(* CODESYS project TcDynCollections.library
   Company: FisoThemes
   DefaultNamespace: TcDynCollections
   Version: 0.1.0.0
   DocFormat: reStructuredText
   Placeholder: TwinCat Dynamic Collections
   Author: Goodwill Mzumala
   Description: A library for handling collections of data dynamically.
   Title: TwinCat Dynamic Collections

Project tree, tasks and I/O mapping:
  libraries: Tc2_Standard, * (Beckhoff Automation GmbH); Tc2_System, * (Beckhoff Automation GmbH); Tc3_Module, * (Beckhoff Automation GmbH)
  DUTs/
    Interfaces/
      interface I_Collections: _Count, _Error_Status, _Is_Empty, Clear
      interface I_List: Add_Front, Create, FB_exit, FB_init, Get, Get_First, Insert, Remove, RemoveAt, Reverse, Set
      interface I_Queue: Dequeue, Dequeue_Void, Enqueue, Enqueue_At_Front, Peek, Reverse
      interface I_Stack: Peek, Pop, Pop_Void, Push, Top
    Structs/
      data type ST_ERROR
      data type ST_NODE
  GVLs/
  POUs/
    Examples/
      program P_List_Example [ST]
      program P_Queue_Example [ST]
      program P_Stack_Example [ST]
    Function Blocks/
      function block FB_Collections [ST]: _Count, _Error_Status, _Is_Empty, Clear
      function block FB_List [ST]: ClearException, EmptyListException, MemCmpErrExpection, OutOfBoundsException, TypeMismatchException, CopyValueTo, DecrementSize, Free_Node, IncrementSize, Iterate, Malloc_Node, SetValue, _Count, _Is_Empty, Add_Front, Clear, Create, FB_exit, FB_init, Get, Get_First, Insert, Remove, RemoveAt, Reverse, Set
      function block FB_Queue [ST]: _Count, _Is_Empty, CatchError, Clear, Dequeue, Dequeue_Void, Enqueue, Enqueue_At_Front, Peek, Reverse
      function block FB_Stack [ST]: _Count, _Is_Empty, CatchError, Clear, Peek, Pop, Pop_Void, Push, Reverse, Top
    program MAIN [ST]
  Project Information/
    function F_GetCompany [ST]
    function F_GetTitle [ST]
    function F_GetVersion [ST]
  UML/
  Version/
    global variables Global_Version
  VISUs/
*)

// DUTs/Structs/ST_ERROR
(* STRUCT used to contain error status information. *)
{attribute 'enable_dynamic_creation'}
TYPE ST_ERROR :
STRUCT
	bSTATUS : BOOL; 		// Indicates if an error has occurred | TRUE = error, FALSE = no error
	nCODE 	: DINT; 		// Error code specific to the particular error.
	sSOURCE : T_MaxString; 	// Textual information describing the error.
END_STRUCT
END_TYPE

// DUTs/Structs/ST_NODE
{attribute 'enable_dynamic_creation'}
TYPE ST_NODE:
STRUCT
	Data 	: __SYSTEM.AnyType; 							// Stored data.
	sData 	: T_MaxString; 									// Data converted to string.
	pNext 	: POINTER TO ST_NODE := Tc3_Module.GVL.NULL; 	// Pointer to next node. (DEFAULT: NULL pointer)
END_STRUCT
END_TYPE

// Version/Global_Version
{attribute 'TcGenerated'}
{attribute 'no-analysis'}
{attribute 'linkalways'}
// This function has been automatically generated from the project information.
VAR_GLOBAL CONSTANT
	{attribute 'const_non_replaced'}
	stLibVersion_TwinCat_Dynamic_Collections : ST_LibVersion := (iMajor := 0, iMinor := 1, iBuild := 0, iRevision := 0, nFlags := 0, sVersion := '0.1.0.0');
END_VAR

// DUTs/Interfaces/I_Collections
INTERFACE I_Collections

(* Number of elements in collection*)
PROPERTY _Count : DINT
GET
END_GET
END_PROPERTY

(* Gets collection's error status *)
PROPERTY _Error_Status : ST_ERROR
GET
END_GET
END_PROPERTY

(* Checks if collection is empty.*)
PROPERTY _Is_Empty : BOOL
GET
END_GET
END_PROPERTY

(* Empties/Clears/Deletes every element on the collection*)
METHOD Clear
END_METHOD

END_INTERFACE

// DUTs/Interfaces/I_List
INTERFACE I_List EXTENDS I_Collections

// Creates/Adds an node to the front of the list
METHOD Add_Front : I_List
VAR_INPUT
	Value 	: ANY; // Value to store in node
END_VAR
END_METHOD

// Creates/Adds an node to the end of the list
METHOD Create : I_List
VAR_INPUT
	Value 	: ANY; // Value to store in node
END_VAR
END_METHOD

METHOD FB_exit : BOOL
VAR_INPUT
	bInCopyCode : BOOL; // if TRUE, the exit method is called for exiting an instance that is copied afterwards (online change).
END_VAR
END_METHOD

METHOD FB_init : BOOL
VAR_INPUT
	bInitRetains : BOOL; // if TRUE, the retain variables are initialized (warm start / cold start)
	bInCopyCode : BOOL;  // if TRUE, the instance afterwards gets moved into the copy code (online change)
END_VAR
END_METHOD

// Gets value from node at specified location;
METHOD Get : I_List
VAR_INPUT
	Return_Value 	: ANY;  // Variable to store requested node value
	nIndex 			: DINT; // Location of node
END_VAR
END_METHOD

(* Gets value from first node. *) 
METHOD Get_First : I_List
VAR_INPUT
	Return_Value 	: ANY; // Variable to store returned value
END_VAR
END_METHOD

// Adds new node to list at specified location
METHOD Insert : I_List
VAR_INPUT
	Value 	: ANY; // Value to store in node
	nIndex 	: DINT; // Location of node
END_VAR
END_METHOD

(* Removes node at the front of the list and returns nothing. *)
METHOD Remove : I_List
END_METHOD

(* Remove node at specific loacation and return nothing *)
METHOD RemoveAt : I_List
VAR_INPUT
	nIndex : DINT; // Location of node
END_VAR
END_METHOD

// Reverses list
METHOD Reverse : I_List
VAR_INPUT
END_VAR
END_METHOD

// Sets value of node at specified location;
METHOD Set : I_List
VAR_INPUT
	Value 	: ANY; 	// Value to store in node
	nIndex 	: DINT; // Location of node
END_VAR
END_METHOD

END_INTERFACE

// DUTs/Interfaces/I_Queue
INTERFACE I_Queue EXTENDS I_Collections

(* Gets and remove item at the front of the queue *)
METHOD Dequeue : I_Queue
VAR_INPUT
	Item : ANY; (* Variable to store returned item value *)
END_VAR
END_METHOD

(* Removes item at the front of the queue without returning anything *)
METHOD Dequeue_Void : I_Queue
VAR_INPUT
END_VAR
END_METHOD

(* Adds item at the back of the queue *)
METHOD Enqueue : I_Queue
VAR_INPUT
	Item : ANY; (* Variable containg data to store on the queue *)
END_VAR
END_METHOD

(* Adds item at the front of the queue *)
METHOD Enqueue_At_Front : I_Queue
VAR_INPUT
	Item : ANY; (* Variable containg data to store on the queue *)
END_VAR
END_METHOD

(* Get item from the queue without removing it. *)
METHOD Peek : I_Queue
VAR_INPUT
	Item 	: ANY; (* Variable to store returned item value *)
	nIndex 	: DINT; (* Location of item*)
END_VAR
END_METHOD

METHOD Reverse : I_Queue
VAR_INPUT
END_VAR
END_METHOD

END_INTERFACE

// DUTs/Interfaces/I_Stack
INTERFACE I_Stack EXTENDS I_Collections

(* Get item from stack without removing it. *)
METHOD Peek : I_Stack
VAR_INPUT
	Item 	: ANY; (* Variable to store returned item value *)
	nIndex 	: DINT; (* Location of item*)
END_VAR
END_METHOD

(* Gets and deletes item at the top of the stack *)
METHOD Pop : I_Stack
VAR_INPUT
	Item : ANY; (* Variable to store returned item value *)
END_VAR
END_METHOD

(* Removes item at the top of the stack without returning anything *)
METHOD Pop_Void : I_Stack
VAR_INPUT
END_VAR
END_METHOD

(* Add item to the top of the stack *)
METHOD Push : I_Stack
VAR_INPUT
	Item : ANY; (* Variable containg data to store on the stack *)
END_VAR
END_METHOD

(* Get item at the top of the stack without removing it. *)
METHOD Top : I_Stack
VAR_INPUT
	Item 	: ANY; (* Variable to store returned item value *)
END_VAR
END_METHOD

END_INTERFACE

// POUs/Examples/P_List_Example
PROGRAM P_List_Example
VAR
	fbList 		: FB_List;
	sData 		: STRING;
	sRTNData	: ARRAY[0..3] OF STRING;
	nCount 		: DINT;
	eState 		: (CREATE, REVERSE, REMOVE, COUNT, IDLE);
	stError 	: ST_ERROR;
END_VAR

stError := fbList._Error_Status;// (stError => stError);
CASE eState OF
	CREATE:
		sData := 'Cats';fbList.Create(sData);
		sData := 'Dogs';fbList.Create(sData);
		sData := 'Birds';fbList.Create(sData);
		sData := 'Fish';fbList.Insert(sData, 1);

		fbList.Get(sRTNData[0], 0)
			  .Get(sRTNData[1], 1)
			  .Get(sRTNData[2], 2)
			  .Get(sRTNData[3], 3);
		eState := IDLE;
	REVERSE:
		fbList.Reverse();
		fbList.Get(sRTNData[0], 0)
			  .Get(sRTNData[1], 1)
			  .Get(sRTNData[2], 2)
			  .Get(sRTNData[3], 3);
		eState := IDLE;
	REMOVE:
		fbList.RemoveAt(2)
			  .Get(sRTNData[0], 0)
			  .Get(sRTNData[1], 1)
			  .Get(sRTNData[2], 2)
			  .Get(sRTNData[3], 3);
		eState := IDLE;
	COUNT: 
		nCount := fbList._Count;
		eState := IDLE;
		
		
END_CASE

END_PROGRAM

// POUs/Function Blocks/FB_List
// Dyanamic List that can store a collection of any types. Similiar to python lists.
FUNCTION_BLOCK FB_List EXTENDS FB_Collections IMPLEMENTS I_List
VAR_INPUT
END_VAR
VAR_OUTPUT
END_VAR
VAR
	
	nSize 		: DINT; // Size of list
	pHead: POINTER TO ST_NODE;
END_VAR

METHOD PROTECTED ClearException : BOOL;
VAR
END_VAR
ClearException 	:= stError.bSTATUS := FALSE;
stError.nCODE 	:= 0;
stError.sSOURCE := 'No error.';
END_METHOD

// Raises an expection if list is empty
METHOD PROTECTED EmptyListException : BOOL
VAR_INPUT
END_VAR
IF THIS^._Is_Empty THEN
	stError.bSTATUS := TRUE;
	stError.nCODE 	:= 2936;
	stError.sSOURCE := 'List is empty';
ELSE
	This^.ClearException();
	END_IF
EmptyListException := stError.bSTATUS;
END_METHOD

// Compares memory sizes of 2 addresses. Returns TRUE  and raises error flag if theyre not same size.
METHOD PROTECTED MemCmpErrExpection : BOOL
VAR_INPUT
	pDestAddr,
	pSrcAddr 	: PVOID;
	nSize 		: UDINT;
END_VAR
VAR_INST
	nMemErr : DINT;
END_VAR
nMemErr := MEMCMP(pDestAddr, pSrcAddr, nSize);
IF nMemErr = -1 THEN 
	stError.bSTATUS := TRUE;
	stError.nCODE 	:= 4129;
	stError.sSOURCE := 'Incorrect parameter values. Destination address smaller than source address';
	
ELSIF nMemErr = 0 THEN THIS^.ClearException();
	
ELSIF nMemErr = 1 THEN
	stError.bSTATUS := TRUE;
	stError.nCODE 	:= 4823;
	stError.sSOURCE := 'Incorrect parameter values. Destination address greater that source address';

ELSE
	stError.bSTATUS := TRUE;
	stError.nCODE 	:= 4564;
	stError.sSOURCE := 'Incorrect parameter values. Pointer to destination/source address is NULL or allocated address memory is NULL.';
	END_IF

MemCmpErrExpection := stError.bSTATUS;
END_METHOD

METHOD PROTECTED OutOfBoundsException : BOOL
VAR_INPUT
	nIndex : DINT;
END_VAR
IF (nIndex < 0) OR (nIndex >= THIS^._Count) THEN
	stError.bSTATUS := TRUE;
	stError.nCODE 	:= 5374;
	stError.sSOURCE := 'Out of bounds. You tried to access data outside the range of this list.';
ELSE
	This^.ClearException();
	END_IF
OutOfBoundsException := stError.bSTATUS;
END_METHOD

METHOD TypeMismatchException : BOOL
VAR_INPUT
	Dest,
	Src 	: __SYSTEM.AnyType;
END_VAR
IF Dest.diSize <> Src.diSize THEN
	stError.bSTATUS := TRUE;
	stError.nCODE 	:= 3172;
	stError.sSOURCE := 'Type mismatch. Byte sizes are not the same';
ELSIF Dest.TypeClass <> Src.TypeClass THEN
	stError.bSTATUS := TRUE;
	stError.nCODE 	:= 3172;
	stError.sSOURCE := 'Type mismatch. Type classes are not the same';
ELSE
	THIS^.ClearException();
END_IF
TypeMismatchException := stError.bSTATUS;
END_METHOD

// Copy data from source memory space to desination memory space
METHOD PROTECTED CopyValueTo
VAR_INPUT
	Dest, Src : __SYSTEM.AnyType;
END_VAR
MEMMOVE(Dest.pValue, Src.pValue, TO_UDINT(Dest.diSize));
END_METHOD

// Decrement list size by 1.
METHOD PROTECTED DecrementSize
VAR_INPUT
END_VAR
THIS^.nSize := THIS^.nSize - 1;
END_METHOD

// Deletes/frees node and it's value from memory
METHOD PROTECTED Free_Node
VAR_INPUT
	pNode : POINTER TO ST_NODE; 
END_VAR
__DELETE(pNode^.Data.pValue);
__DELETE(pNode);
END_METHOD

// Increments list size by 1
METHOD PROTECTED IncrementSize
VAR_INPUT
END_VAR
THIS^.nSize := THIS^.nSize + 1;
END_METHOD

// Returns pointer to node at specificied location;
METHOD PROTECTED Iterate : POINTER TO ST_NODE
VAR_INPUT
	nIndex : DINT;
END_VAR
VAR 
	i 		: DINT;
	pTemp 	: POINTER TO ST_NODE;
END_VAR
IF THIS^.OutOfBoundsException(nIndex) THEN RETURN; END_IF
IF nIndex = 0 THEN Iterate := THIS^.pHead; RETURN; END_IF
//IF nIndex = THIS^._Count-1 THEN Iterate := pTail; RETURN; END_IF
pTemp := pHead;
FOR i := 1 TO nIndex DO pTemp := pTemp^.pNext; END_FOR
Iterate := pTemp;
END_METHOD

// Allocate memory space for node and the value for it's data on the heap, returns pointer to node;
// WARNING!!! Always have a place to store the node pointer otherwise a memory leak will occur.
METHOD PROTECTED Malloc_Node : POINTER TO ST_NODE
VAR_INPUT
	Variable : __SYSTEM.AnyType;
END_VAR
VAR
	pTemp 	: POINTER TO ST_NODE;
END_VAR
pTemp := __NEW(ST_NODE); // Allocate space in memory for a node.
pTemp^.Data := Variable;
pTemp^.Data.pValue := __NEW(BYTE, TO_UDINT(Variable.diSize)); // Allocate space in memory to store data value.
Malloc_Node := pTemp;
END_METHOD

(* Set value of __SYSTEM.Anytype variable *)
METHOD PROTECTED SetValue
VAR_INPUT
	Variable	: __SYSTEM.Anytype;
	Value 		: USINT; // Character/byte to set.
END_VAR
MEMSET(Variable.pValue, Value, TO_UDINT(Variable.diSize));
END_METHOD

// Number of elements in list
PROPERTY PUBLIC _Count : DINT
GET
_Count := nSize;
END_GET
END_PROPERTY

(* Checks of list is empty.*)
PROPERTY _Is_Empty : BOOL
GET
_Is_Empty := (THIS^._Count = 0) AND (THIS^.pHead = 0);
END_GET
END_PROPERTY

// Creates/Adds an node to the front of the list
METHOD Add_Front : I_List
VAR_INPUT
	Value 	: ANY; // Value to store in node
END_VAR
VAR
	pTemp 	: POINTER TO ST_NODE;
END_VAR
Add_Front := THIS^;
pTemp := THIS^.Malloc_Node(Value);
THIS^.CopyValueTo(pTemp^.Data, Value);

pTemp^.pNext := THIS^.pHead; THIS^.pHead := pTemp;
THIS^.IncrementSize();
END_METHOD

(* Empties/Clears/Deletes every node on the list*)
METHOD Clear
VAR
	pTemp : POINTER TO ST_NODE;
END_VAR
pTemp := THIS^.pHead;
WHILE pTemp <> 0 DO
	pTemp := pTemp^.pNext; THIS^.Remove();
END_WHILE
END_METHOD

// Creates/Adds an node to the end of the list
METHOD Create : I_List
VAR_INPUT
	Value 	: ANY; // Value to store in node
END_VAR
VAR
	pTemp 	: POINTER TO ST_NODE;
END_VAR
Create := THIS^;
pTemp := THIS^.Malloc_Node(Value);
THIS^.CopyValueTo(pTemp^.Data, Value);

IF THIS^._Is_Empty THEN THIS^.pHead := pTemp;
ELSE Iterate(THIS^._Count - 1)^.pNext := pTemp; END_IF

THIS^.IncrementSize();
END_METHOD

METHOD FB_exit : BOOL
VAR_INPUT
	(* if TRUE, the exit method is called for exiting an instance that is copied afterwards (online change).*)
	bInCopyCode	: BOOL;
END_VAR
This^.Clear();
END_METHOD

METHOD FB_init : BOOL
VAR_INPUT
	bInitRetains : BOOL; // if TRUE, the retain variables are initialized (warm start / cold start)
	bInCopyCode : BOOL;  // if TRUE, the instance afterwards gets moved into the copy code (online change)
END_VAR
THIS^.Clear();
THIS^.pHead := Tc3_Module.GVL.NULL;
END_METHOD

(* Gets value from node at specified location;*)
METHOD Get : I_List
VAR_INPUT
	Return_Value 	: ANY;(* Variable to store requested node value*)
	nIndex			: DINT; (* Location of node*)
END_VAR
VAR
	pTemp : POINTER TO ST_NODE;
END_VAR
Get := THIS^;
IF THIS^.EmptyListException() OR THIS^.OutOfBoundsException(nIndex) THEN THIS^.SetValue(Return_Value, 16#0); RETURN; END_IF
pTemp := Iterate(nIndex);
IF THIS^.TypeMismatchException(Return_Value, pTemp^.Data) THEN THIS^.SetValue(Return_Value, 16#0); RETURN; END_IF
THIS^.CopyValueTo(Return_Value, pTemp^.Data);
END_METHOD

(* Gets value from first node. *)
METHOD Get_First : I_List
VAR_INPUT
	Return_Value : ANY; // Variable to store returned value
END_VAR
VAR
	pTemp 	: POINTER TO ST_NODE;
END_VAR
Get_First := THIS^;
IF THIS^.TypeMismatchException(Return_Value, pHead^.Data) OR THIS^.EmptyListException() THEN THIS^.SetValue(Return_Value, 16#0); RETURN; END_IF
THIS^.CopyValueTo(Return_Value, pHead^.Data);
Get_First := THIS^;
END_METHOD

(* Adds new node to list at specified location*)
METHOD Insert : I_List
VAR_INPUT
	Value	: ANY;(* Value to store in node*)
	nIndex	: DINT;(* Location of node*)
END_VAR
VAR
	pPrevious 	: POINTER TO ST_NODE;
	pCurrent 	: POINTER TO ST_NODE;
	pTemp 		: POINTER TO ST_NODE;
END_VAR
Insert := THIS^;
IF nIndex = THIS^._Count THEN THIS^.Create(Value); END_IF
IF THIS^.OutOfBoundsException(nIndex) THEN RETURN; END_IF
IF nIndex = 0 THEN THIS^.Add_Front(Value); RETURN; END_IF

pTemp := THIS^.Malloc_Node(Value);
THIS^.CopyValueTo(pTemp^.Data, Value);

pPrevious := THIS^.Iterate(nIndex-1);
pCurrent := pPrevious^.pNext;
pPrevious^.pNext := pTemp;
pTemp^.pNext := pCurrent;

THIS^.IncrementSize();
END_METHOD

(* Removes node at the front of the list and returns nothing. *)
METHOD Remove : I_List
VAR
	pTemp 	: POINTER TO ST_NODE;
END_VAR
Remove := THIS^;
IF THIS^._Is_Empty THEN RETURN; END_IF

pTemp := THIS^.pHead^.pNext;
THIS^.Free_Node(pHead);
THIS^.pHead := pTemp;

THIS^.DecrementSize();
END_METHOD

(* Remove node at specific loacation and return nothing *)
METHOD RemoveAt : I_List
VAR_INPUT
	nIndex	: DINT;(* Location of node*)
END_VAR
VAR
	pTemp : ARRAY[1..2] OF POINTER TO ST_NODE;
END_VAR
RemoveAt := THIS^;
IF THIS^.EmptyListException() OR THIS^.OutOfBoundsException(nIndex)  THEN RETURN; END_IF
IF nIndex = 0 THEN THIS^.Remove(); RETURN; END_IF

pTemp[1] := THIS^.Iterate(nIndex-1);
pTemp[2] := pTemp[1]^.pNext^.pNext;
THIS^.Free_Node(pTemp[1]^.pNext);
pTemp[1]^.pNext := pTemp[2];

THIS^.DecrementSize();
END_METHOD

(* Reverses list*)
METHOD Reverse : I_List
VAR
	pPrevious 	: POINTER TO ST_NODE;
	pCurrent 	: POINTER TO ST_NODE;
	pNext	 	: POINTER TO ST_NODE;
END_VAR
Reverse := THIS^;
pCurrent := pHead;
WHILE pCurrent <> 0 DO
	pNext := pCurrent^.pNext;
	pCurrent^.pNext := pPrevious;
	pPrevious := pCurrent;
	pCurrent := pNext;
END_WHILE
THIS^.pHead := pPrevious;
END_METHOD

(* Sets value of node at specified location;*)
METHOD Set : I_List
VAR_INPUT
	Value	: ANY; (* Value to store in node*)
	nIndex	: DINT; (* Location of node*)
END_VAR
VAR
	pTemp : POINTER TO ST_NODE;
END_VAR
Set := THIS^;
IF THIS^.OutOfBoundsException(nIndex) THEN RETURN; END_IF
pTemp := Iterate(nIndex);
IF THIS^.TypeMismatchException(pTemp^.Data, Value) THEN RETURN; END_IF
THIS^.CopyValueTo(pTemp^.Data, Value);
END_METHOD

END_FUNCTION_BLOCK

// POUs/Function Blocks/FB_Collections
FUNCTION_BLOCK ABSTRACT FB_Collections IMPLEMENTS I_Collections
VAR_INPUT
END_VAR
VAR_OUTPUT
END_VAR
VAR
	stError : ST_ERROR;
END_VAR

(* Number of elements in collection*)
PROPERTY _Count : DINT
GET
END_GET
END_PROPERTY

(* Gets collection's error status *)
PROPERTY _Error_Status : ST_ERROR
GET
_Error_Status := THIS^.stError;
END_GET
END_PROPERTY

(* Checks if collection is empty.*)
PROPERTY _Is_Empty : BOOL
GET
END_GET
END_PROPERTY

(* Empties/Clears/Deletes every element on the collection*)
METHOD Clear
END_METHOD

END_FUNCTION_BLOCK

// POUs/Examples/P_Queue_Example
// Login into PLC and live write eState. Try nData and nRTNData once your done. eState Initialises at IDLE
PROGRAM P_Queue_Example
VAR
	fbList 		: FB_LIST;
	fbQueue 	: FB_Queue;
	sData 		: STRING;
	sRTNData	: ARRAY[0..3] OF STRING; //returned data
	nData 		: DINT;
	nRTNData 	: ARRAY[0..3] OF DINT; 
	nCount 		: DINT;
	eState 		: (IDLE, ENQUEUE_AND_PEEK, GET_ITEM_COUNT,REVERSE_AND_PEEK, DEQUEUE_AND_PEEK, CLEAR_Q);
	stError 	: ST_ERROR;
END_VAR

fbQueue(ipList := fbList);
stError := fbQueue._Error_Status;
CASE eState OF
	ENQUEUE_AND_PEEK: //
		sData := 'Cats';fbQueue.Enqueue(sData);
		sData := 'Dogs';fbQueue.Enqueue(sData);
		sData := 'Birds';fbQueue.Enqueue(sData);
		sData := 'Fish';fbQueue.Enqueue_At_Front(sData);

		fbQueue.Peek(sRTNData[0], 0)
			   .Peek(sRTNData[1], 1)
			   .Peek(sRTNData[2], 2)
			   .Peek(sRTNData[3], 3);
		eState := IDLE;
		
	GET_ITEM_COUNT: 
		nCount := fbQueue._Count;
		eState := IDLE;
		
	REVERSE_AND_PEEK:
		fbQueue.Reverse()
			   .Peek(sRTNData[0], 0)
			   .Peek(sRTNData[1], 1)
			   .Peek(sRTNData[2], 2)
			   .Peek(sRTNData[3], 3);
		eState := IDLE;
	
	DEQUEUE_AND_PEEK:
		fbQueue.Dequeue(sRTNData[0])
			   .Dequeue_Void()
			   .Peek(sRTNData[1], 1)
			   .Peek(sRTNData[2], 2)
			   .Peek(sRTNData[3], 3);
		eState := IDLE;
		
	CLEAR_Q:
		fbQueue.Clear();
		eState := IDLE;	
END_CASE

END_PROGRAM

// POUs/Function Blocks/FB_Queue
FUNCTION_BLOCK FB_Queue EXTENDS FB_Collections  IMPLEMENTS I_Queue
VAR_INPUT
	ipList : I_List; // List to perform operations on.
END_VAR
VAR
	//ipItems_List : I_List; // List holding items on the queue
END_VAR

(* Number of items in queue*)
PROPERTY _Count : DINT
GET
_Count := THIS^.ipList._Count;
END_GET
END_PROPERTY

(* Checks of queue is empty.*)
PROPERTY _Is_Empty : BOOL
GET
_Is_Empty := THIS^.ipList._Is_Empty;
END_GET
END_PROPERTY

METHOD PROTECTED CatchError : BOOL
VAR_INPUT
END_VAR
//THIS^.ipItems_List(stError => THIS^.stError);
THIS^.stError := ipList._Error_Status;
CatchError := stError.bSTATUS;
END_METHOD

(* Empties/Clears/Deletes every item on the queue*)
METHOD Clear
THIS^.ipList.Clear();
END_METHOD

(* Gets and remove item at the front of the queue *)
METHOD Dequeue : I_Queue
VAR_INPUT
	Item : ANY; (* Variable to store returned item value *)
END_VAR
Dequeue := THIS^;
THIS^.ipList.Get_First(Item);
IF THIS^.CatchError() THEN RETURN; END_IF;
THIS^.ipList.Remove();
THIS^.CatchError();
END_METHOD

(* Removes item at the front of the queue without returning anything *)
METHOD Dequeue_Void : I_Queue
VAR_INPUT
END_VAR
Dequeue_Void := THIS^;
THIS^.ipList.Remove();
THIS^.CatchError();
END_METHOD

(* Adds item at the back of the queue *)
METHOD Enqueue : I_Queue
VAR_INPUT
	Item : ANY; (* Variable containg data to store on the queue *)
END_VAR
Enqueue := THIS^;
THIS^.ipList.Create(Item);
THIS^.CatchError();
END_METHOD

(* Adds item at the front of the queue *)
METHOD Enqueue_At_Front : I_Queue
VAR_INPUT
	Item : ANY; (* Variable containg data to store on the queue *)
END_VAR
Enqueue_At_Front := THIS^;
THIS^.ipList.Add_Front(Item);
THIS^.CatchError();
END_METHOD

(* Get item from the queue without removing it. *)
METHOD Peek : I_Queue
VAR_INPUT
	Item 	: ANY; (* Variable to store returned item value *)
	nIndex 	: DINT; (* Location of item*)
END_VAR
Peek := THIS^;
THIS^.ipList.Get(Item, nIndex);
THIS^.CatchError();
END_METHOD

METHOD Reverse : I_Queue
VAR_INPUT
END_VAR
Reverse := THIS^;
THIS^.ipList.Reverse();
THIS^.CatchError();
END_METHOD

END_FUNCTION_BLOCK

// POUs/Examples/P_Stack_Example
// Login into PLC and live write eState. Try nData and nRTNData once your done. eState Initialises at IDLE
PROGRAM P_Stack_Example
VAR
	fbList 		: FB_LIST;
	fbStack 	: FB_Stack;
	sData 		: STRING;
	sRTNData	: ARRAY[0..3] OF STRING; //returned data
	nData 		: DINT;
	nRTNData 	: ARRAY[0..3] OF DINT; 
	nCount 		: DINT;
	eState 		: (IDLE, PUSH_AND_PEEK, GET_ITEM_COUNT,REVERSE_AND_PEEK, POP, CLEAR_STACK);
	stError 	: ST_ERROR;
END_VAR

fbStack(ipList := fbList);
stError := fbStack._Error_Status;
CASE eState OF
	PUSH_AND_PEEK:
		sData := 'Cats';fbStack.Push(sData);
		sData := 'Dogs';fbStack.Push(sData);
		sData := 'Birds';fbStack.Push(sData);
		sData := 'Fish';fbStack.Push(sData);

		fbStack.Peek(sRTNData[0], 0)
			   .Peek(sRTNData[1], 1)
			   .Peek(sRTNData[2], 2)
			   .Peek(sRTNData[3], 3);
		eState := IDLE;
		
	GET_ITEM_COUNT: 
		nCount := fbStack._Count;
		eState := IDLE;
		
	REVERSE_AND_PEEK:
		fbStack.Reverse()
			   .Peek(sRTNData[0], 0)
			   .Peek(sRTNData[1], 1)
			   .Peek(sRTNData[2], 2)
			   .Peek(sRTNData[3], 3);
		eState := IDLE;
	
	POP:
		fbStack.Pop(sRTNData[0])
			   .Pop(sRTNData[1])
			   .Pop(sRTNData[2]);
		eState := IDLE;
		
	CLEAR_STACK:
		fbStack.Clear();
		eState := IDLE;	
END_CASE

END_PROGRAM

// POUs/Function Blocks/FB_Stack
FUNCTION_BLOCK FB_Stack EXTENDS FB_Collections IMPLEMENTS I_Stack
VAR_INPUT
	ipList : I_List; // List to perform operations on.
END_VAR
VAR_OUTPUT
END_VAR

(* Number of elements in the stack *)
PROPERTY _Count : DINT
GET
_Count := THIS^.ipList._Count;
END_GET
END_PROPERTY

(* Checks of stack is empty.*)
PROPERTY _Is_Empty : BOOL
GET
_Is_Empty := THIS^.ipList._Is_Empty;
END_GET
END_PROPERTY

METHOD PROTECTED CatchError : BOOL
VAR_INPUT
END_VAR
stError := THIS^.ipList._Error_Status;
CatchError := stError.bSTATUS;
END_METHOD

(* Empties/Clears/Deletes every item on the stack*)
METHOD Clear
VAR_INPUT
END_VAR
THIS^.ipList.Clear();
END_METHOD

(* Get item from stack without removing it. *)
METHOD Peek : I_Stack
VAR_INPUT
	Item 	: ANY; (* Variable to store returned item value *)
	nIndex 	: DINT; (* Location of item*)
END_VAR
Peek := THIS^;
THIS^.ipList.Get(Item, nIndex);
THIS^.CatchError();
END_METHOD

(* Gets and deletes item at the top of the stack *)
METHOD Pop : I_Stack
VAR_INPUT
	Item : ANY; (* Variable to store returned item value *)
END_VAR
Pop := THIS^;
THIS^.ipList.Get_First(Item);
IF THIS^.CatchError() THEN RETURN; END_IF;
THIS^.ipList.Remove();
THIS^.CatchError();
END_METHOD

(* Removes item at the top of the stack without returning anything *)
METHOD Pop_Void : I_Stack
VAR_INPUT
END_VAR
Pop_Void := THIS^;
THIS^.ipList.Remove();
THIS^.CatchError();
END_METHOD

(* Add item to the top of the stack *)
METHOD Push : I_Stack
VAR_INPUT
	Item : ANY; (* Variable containg data to store on the stack *)
END_VAR
Push := THIS^;
THIS^.ipList.Add_Front(Item);
THIS^.CatchError();
END_METHOD

(* Reverses order of items on stack *)
METHOD Reverse : I_Stack
VAR_INPUT
END_VAR
Reverse := THIS^;
THIS^.ipList.Reverse();
THIS^.CatchError();
END_METHOD

(* Get item at the top of the stack without removing it. *)
METHOD Top : I_Stack
VAR_INPUT
	Item 	: ANY; (* Variable to store returned item value *)
END_VAR
Top := THIS^;
THIS^.ipList.Get_First(Item);
IF THIS^.CatchError() THEN RETURN; END_IF;
END_METHOD

END_FUNCTION_BLOCK

// POUs/MAIN
PROGRAM MAIN
VAR
END_VAR

P_List_Example();
P_Queue_Example();
P_Stack_Example();

END_PROGRAM

// Project Information/F_GetCompany
// This function has been automatically generated from the project information.
{attribute 'signature_flag' := '1073741824'}
{attribute 'TcGenerated'}
{attribute 'no-analysis'}
FUNCTION F_GetCompany : WSTRING
VAR_INPUT
	
END_VAR

F_GetCompany := "FisoThemes";

END_FUNCTION

// Project Information/F_GetTitle
// This function has been automatically generated from the project information.
{attribute 'signature_flag' := '1073741824'}
{attribute 'TcGenerated'}
{attribute 'no-analysis'}
FUNCTION F_GetTitle : WSTRING
VAR_INPUT
	
END_VAR

F_GetTitle := "TwinCat Dynamic Collections";

END_FUNCTION

// Project Information/F_GetVersion
// This function has been automatically generated from the project information.
{attribute 'signature_flag' := '1073741824'}
{attribute 'TcGenerated'}
{attribute 'no-analysis'}
FUNCTION F_GetVersion : ST_LibVersion
VAR_INPUT
	
END_VAR

F_GetVersion.iMajor := 0;
F_GetVersion.iMinor := 1;
F_GetVersion.iBuild := 0;
F_GetVersion.iRevision := 0;

END_FUNCTION
